% RSLogix 500 project O2 concentration.RSS, saved by version 8.30.00.16 %
PROJECT "UNTITLED"    % processor: Bul.1763 MicroLogix 1100 Series B %

PROGRAM FILES
  LAD 2 "MAIN"  2 rungs
  LAD 3 "I/O"  11 rungs

DATA FILES
  O0 OUTPUT  6 elements
  I1 INPUT  12 elements
  S2 STATUS  66 elements
  B3 BINARY  1 elements
  T4 TIMER  4 elements
  C5 COUNTER  2 elements
  R6 CONTROL  1 elements
  N7 INTEGER  4 elements
  F8 FLOAT  9 elements

LADDER 2 "MAIN"
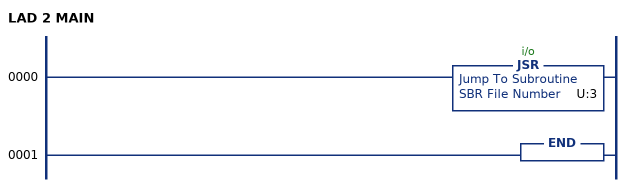
% Rung: 0 %
SOR JSR U:3 EOR
%   U:3  "i/o" %
% Rung: 1 %
SOR END EOR

LADDER 3 "I/O"
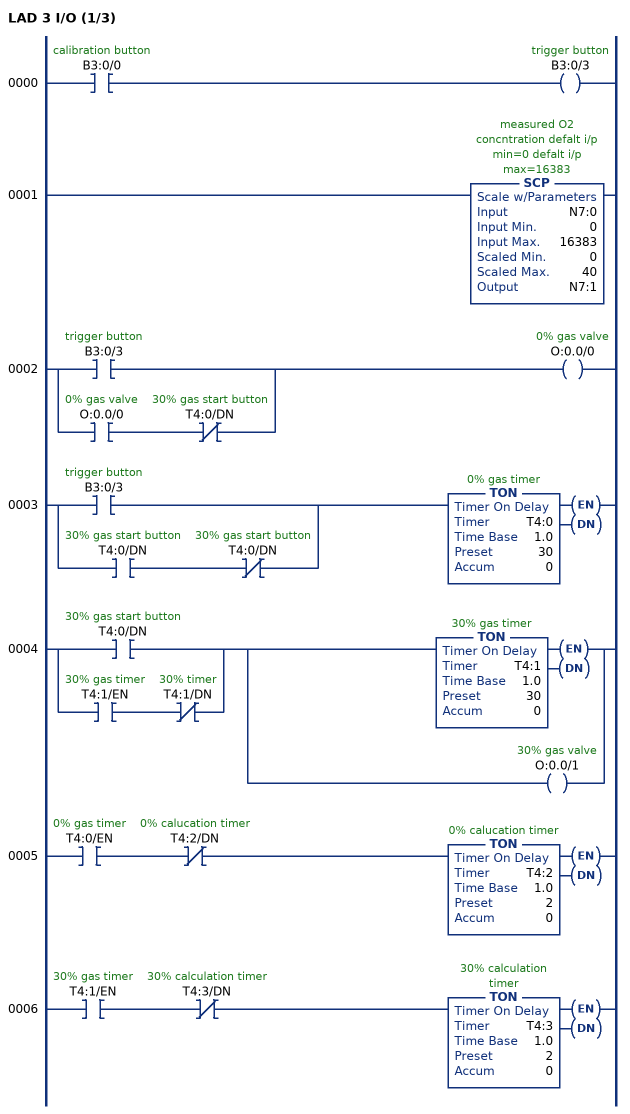
% Rung: 0 %
SOR XIC B3:0/0 OTE B3:0/3 EOR
%   B3:0/0  "calibration button" %
%   B3:0/3  "trigger button" %
% Rung: 1 %
SOR SCP N7:0 0 16383 0 40 N7:1 EOR
%   N7:0  "O2 sensor input signal" %
%   N7:1  "measured O2 concntration defalt i/p min=0 defalt i/p max=16383" %
% Rung: 2 %
SOR BST XIC B3:0/3 NXB XIC O:0.0/0 XIO T4:0/DN BND OTE O:0.0/0 EOR
%   B3:0/3  "trigger button" %
%   O:0.0/0  "0% gas valve" %
%   T4:0/DN  "30% gas start button" %
% Rung: 3 %
SOR BST XIC B3:0/3 NXB XIC T4:0/DN XIO T4:0/DN BND TON T4:0 1.0 30 0 EOR
%   B3:0/3  "trigger button" %
%   T4:0/DN  "30% gas start button" %
%   T4:0  "0% gas timer" %
% Rung: 4 %
SOR BST XIC T4:0/DN NXB XIC T4:1/EN XIO T4:1/DN BND BST TON T4:1 1.0 30 0 NXB OTE O:0.0/1 BND EOR
%   T4:0/DN  "30% gas start button" %
%   T4:1  "30% gas timer" %
%   T4:1/DN  "30% timer" %
%   O:0.0/1  "30% gas valve" %
% Rung: 5 %
SOR XIC T4:0/EN XIO T4:2/DN TON T4:2 1.0 2 0 EOR
%   T4:0  "0% gas timer" %
%   T4:2  "0% calucation timer" %
% Rung: 6 %  % edit flag set %
SOR XIC T4:1/EN XIO T4:3/DN TON T4:3 1.0 2 0 EOR
%   T4:1  "30% gas timer" %
%   T4:3  "30% calculation timer" %

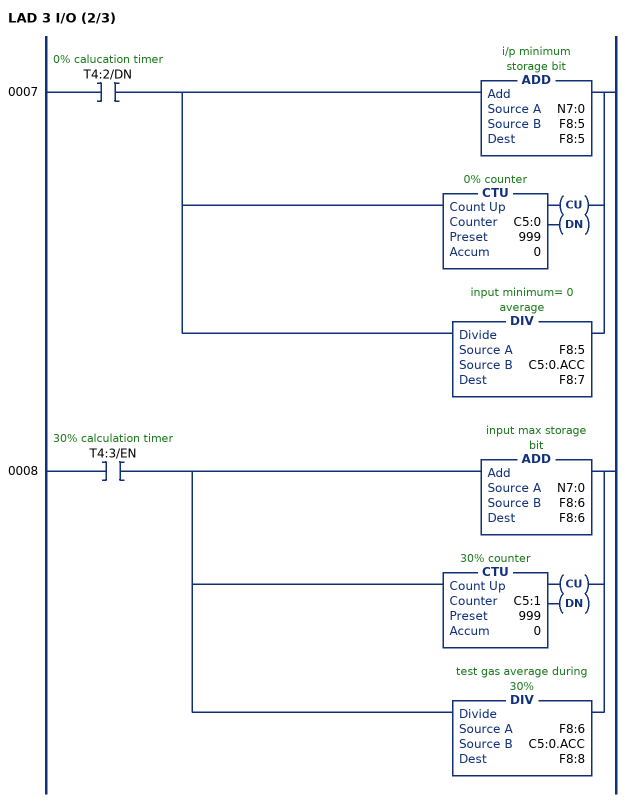
% Rung: 7 %
SOR XIC T4:2/DN BST ADD N7:0 F8:5 F8:5 NXB CTU C5:0 999 0 NXB DIV F8:5 C5:0.ACC F8:7 BND EOR
%   T4:2  "0% calucation timer" %
%   N7:0  "O2 sensor input signal" %
%   F8:5  "i/p minimum storage bit" %
%   C5:0  "0% counter" %
%   F8:7  "input minimum= 0 average" %
% Rung: 8 %
SOR XIC T4:3/EN BST ADD N7:0 F8:6 F8:6 NXB CTU C5:1 999 0 NXB DIV F8:6 C5:0.ACC F8:8 BND EOR
%   T4:3  "30% calculation timer" %
%   N7:0  "O2 sensor input signal" %
%   F8:6  "input max storage bit" %
%   C5:1  "30% counter" %
%   C5:0  "0% counter" %
%   F8:8  "test gas average during 30%" %

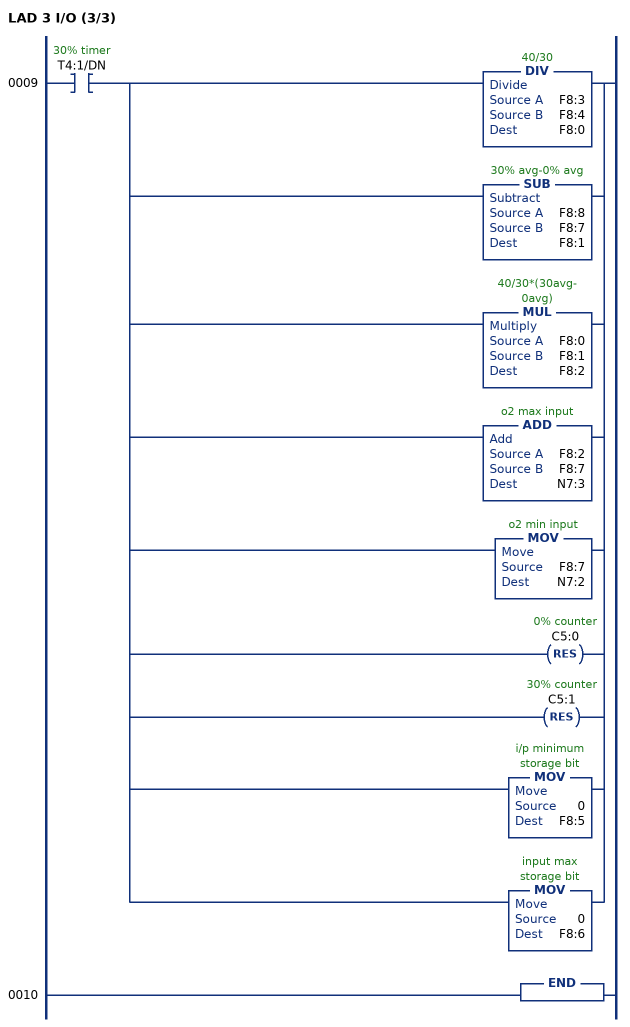
% Rung: 9 %
SOR XIC T4:1/DN BST DIV F8:3 F8:4 F8:0 NXB SUB F8:8 F8:7 F8:1 NXB MUL F8:0 F8:1 F8:2 NXB ADD F8:2 F8:7 N7:3 NXB MOV F8:7 N7:2 NXB RES C5:0 NXB RES C5:1 NXB MOV 0 F8:5 NXB MOV 0 F8:6 BND EOR
%   T4:1/DN  "30% timer" %
%   F8:3  "40" %
%   F8:4  "30" %
%   F8:0  "40/30" %
%   F8:8  "test gas average during 30%" %
%   F8:7  "input minimum= 0 average" %
%   F8:1  "30% avg-0% avg" %
%   F8:2  "40/30*(30avg-0avg)" %
%   N7:3  "o2 max input" %
%   N7:2  "o2 min input" %
%   C5:0  "0% counter" %
%   C5:1  "30% counter" %
%   F8:5  "i/p minimum storage bit" %
%   F8:6  "input max storage bit" %
% Rung: 10 %
SOR END EOR

OTHER DOCUMENTED ADDRESSES
  B3:0/1  "0% gas valve bit"
  B3:0/2  "30% gas valve bit"

DATA TABLE (non-zero values as saved)
DATA T4
% .PRE .ACC %
% T4:0 % 30 0
% T4:1 % 30 0
% T4:2 % 2 0
% T4:3 % 2 0
DATA C5
% .PRE .ACC %
% C5:0 % 999 0
% C5:1 % 999 0
